TYPE "CoilHandling_Config"
VERSION : 0.1
// Block: CoilHandling_Config
   STRUCT
      SensorsDelayOn : Time;
      SensorsDelayOff : Time;
      CoilDiameterSetLoopSynchro : Real;
      CoilDiameterRstLoopSynchro : Real;
      MatCounter_Exist : Bool;
   END_STRUCT;

END_TYPE
